FUNCTION_BLOCK Machine EXTENDS FB_PackML_BaseModule
VAR
	EquipOne	: EquipmentModule := (Name := 'Equip One');
	EquipTwo	: EquipmentModuleWithSubModule := (Name := 'Equip Two');
	ComponentMM : Component		  := (Name := 'Component MM');

	//Alarms
	MachineAlarms : ARRAY[1..MACHINE_ALARM_COUNT] OF FB_TcAlarm;
	testCritical  : BOOL;
	testError	  : BOOL;
	testWarning	  : BOOL;
	testInfo	  : BOOL;
	testVerbose	  : BOOL;
	clearAlarms	  : BOOL;
END_VAR

VAR CONSTANT
	MACHINE_ALARM_COUNT : UDINT := 6; //First is InitReferenceEvent
END_VAR

METHOD PROTECTED Clearing
VAR
	i				: UDINT;
	SubModulesReady : BOOL := TRUE;
	ComponentsReady : BOOL := TRUE;
END_VAR
(*
If there are no Components of the Machine
then we can clear the Machine Alarms and let the SUPER handle the rest.

But if the Machine Module has a component
then the process of clearing the alarms 
must be handled in a slightly different manner.
This will prevent an existing alarm condition that is still TRUE
from being cleared and raised multiple times.
*)
IF NumberOfComponents = 0 THEN
	F_ClearAllEventsInClass(Alarms := MachineAlarms);
	SUPER^.Clearing();
ELSE
	CASE SequenceState OF
		0:
			F_ClearAllEventsInClass(Alarms := MachineAlarms);
			SequenceState := SequenceState + 10;

		10:
			FOR i := 1 TO NumberOfSubModules DO
				ipSubModules[i].StateCommand := ePMLCommand_Clear;
			END_FOR

			IF BaseAlarms[E_BaseAlarms.ComponentError].bRaised THEN
				BaseAlarms[E_BaseAlarms.ComponentError].Clear(0, 0);
			END_IF;

			IF BaseAlarms[E_BaseAlarms.SubModuleError].bRaised THEN
				BaseAlarms[E_BaseAlarms.SubModuleError].Clear(0, 0);
			END_IF;

			SequenceState := SequenceState + 10;

		20:
			FOR i := 1 TO NumberOfComponents DO
				IF Parameters_PackML_Base.RESET_COMPONENTS_WITHOUT_ERROR THEN
					ipComponents[i].Reset();
				ELSE
					IF ipComponents[i].Error THEN
						ipComponents[i].Reset();
					END_IF
				END_IF
			END_FOR

			FOR i := 1 TO NumberOfComponents DO
				ComponentsReady := ComponentsReady AND NOT ipComponents[i].Error;
			END_FOR

			IF ComponentsReady THEN
				SequenceState := SequenceState + 10;
			END_IF

		30:
			FOR i := 1 TO NumberOfSubModules DO
				SubModulesReady := SubModulesReady AND (ipSubModules[i].CurrentState = ePMLState_Stopped);
			END_FOR

			IF SubModulesReady AND (StateTasksComplete OR NoStateTasksToComplete) THEN
				NoStateTasksToComplete := TRUE;
				StateTasksComplete	   := FALSE;
				StateComplete();
			END_IF
	END_CASE
END_IF
END_METHOD

//! @summary Initializes event function blocks using this module's name
METHOD PROTECTED CreateEvents

//! @description This method is called by <c>Initialize()</c> as required
F_CreateAllEventsInClass(Alarms		:= MachineAlarms,
						 ClassSize	:= SIZEOF(TC_Events.MachineEvents),
						 pInitEvent := ADR(TC_EVENTS.MachineEvents.InitReferenceEvent),
						 Prefix		:= Name);

SUPER^.CreateEvents();
END_METHOD

//! @summary This method serves as the entry point for all underlying FB logic

//! @description This method should be called cyclically by descendant function blocks by invoking <c>SUPER^.CyclicLogic()</c>.  Alternatively, the contents of this method could be reimplemented entirely in which case a call to this method would not be necessary.
METHOD PUBLIC CyclicLogic
VAR
	i : UDINT;
END_VAR
IF NOT _InitComplete THEN
	_InitComplete := Initialize();
	RETURN;
END_IF

//AlarmHandling();
IF testVerbose AND NOT MachineAlarms[E_MachineEvents.VerboseEvent].bRaised THEN
	RaiseAlarm2Args(MachineAlarms[E_MachineEvents.VerboseEvent], 'Note 1', 'Note 2');
END_IF

IF testCritical AND NOT MachineAlarms[E_MachineEvents.CriticalEvent].bRaised THEN
	RaiseAlarm2Args(MachineAlarms[E_MachineEvents.CriticalEvent], 'Note 1', 'Note 2');
END_IF

//The MachineMonitor is based on the SubModuleMonitor, but is only monitors itself
MachineMonitor();

//
SUPER^.CyclicLogic();

(*
*
*		Code must be after SUPER^.CyclicLogic();
*
*)

(* Update alarm severity from this module *)
_CurrentAlarmSeverity := F_GetMaxSeverityRaised(Alarms := MachineAlarms, CurrentSeverity := _CurrentAlarmSeverity);
_Error				  := _CurrentAlarmSeverity >= TcEventSeverity.Error;


Trace(Message:='Test Mesage');
END_METHOD

//! @summary Basic module initialization logic
METHOD PROTECTED Initialize : BOOL;
VAR
	i						 : UDINT;
	varInfo					 : __SYSTEM.VAR_INFO;
	AllSubUnitsInitialized	 : BOOL := TRUE;
	AllComponentsInitialized : BOOL := TRUE;
END_VAR

//! @description This method is called by <c>CyclicLogic()</c> as required
Initialize := FALSE;
CASE DescendantSequenceState OF
	0:
		LogModeChanges	:= FALSE;
		LogStateChanges := FALSE;

		//Register Submodules
		RegisterSubmodule(EquipOne);
		RegisterSubmodule(EquipTwo);		
		RegisterComponent(ComponentMM);
		DescendantSequenceState := DescendantSequenceState + 10;

	10:
		IF SUPER^.Initialize() THEN
			Initialize := TRUE;
		END_IF
END_CASE
END_METHOD

METHOD MachineMonitor
VAR
	AlarmResponses : ARRAY[0..4] OF E_AlarmResponse; //Temporary response array	
	i			   : UDINT;
END_VAR
IF _CurrentState <> E_PMLState.ePMLState_Aborted AND _CurrentState <> E_PMLState.ePMLState_Aborting AND _CurrentState <> E_PMLState.ePMLState_Clearing AND _CurrentState <> E_PMLState.ePMLState_Stopped AND _CurrentState <> E_PMLState.ePMLState_Stopping THEN
	AlarmResponses := ParentResponseDefinitions;
	CASE AlarmResponses[_CurrentAlarmSeverity] OF
		E_AlarmResponse.Abort_ImmediateError:
			AbortImmediateError(Name, TRUE);

		E_AlarmResponse.Abort_Immediate:
			AbortImmediate();

		E_AlarmResponse.Stop_Immediate:
			StopImmediate();

		E_AlarmResponse.Stop_Controlled:
			StopControlled();

		E_AlarmResponse.Hold_Immediate:
			HoldImmediate();

		E_AlarmResponse.Hold_Controlled:
			HoldControlled();

		E_AlarmResponse.Suspend_Immediate:
			SuspendImmediate();

		E_AlarmResponse.Suspend_Controlled:
			SuspendControlled();

		E_AlarmResponse.NoResponse:
			;
	END_CASE
ELSIF _CurrentState = E_PMLState.ePMLState_Stopped OR _CurrentState = E_PMLState.ePMLState_Stopping THEN
	AlarmResponses := ParentResponseDefinitions;
	CASE AlarmResponses[CurrentAlarmSeverity] OF
		E_AlarmResponse.Abort_ImmediateError:
			AbortImmediateError(Name, TRUE);

		E_AlarmResponse.Abort_Immediate:
			AbortImmediate();

		E_AlarmResponse.NoResponse:
			;
	END_CASE
END_IF
END_METHOD

METHOD RaiseAlarm2Args
VAR_IN_OUT
	Alarm : FB_TcAlarm; //Alarm to be raised
END_VAR

VAR_INPUT
	String_1 : STRING; //First String Parameter (The Name of this component will be applied first automatically)
	String_2 : STRING; //Second String Parameter
END_VAR
F_RaiseAlarmWithStringParameters(Alarm	  := Alarm,
								 String_1 := Name,
								 String_2 := String_1,
								 String_3 := String_2);
END_METHOD

END_FUNCTION_BLOCK

(* stored: Version 1.1.0.1, ProductVersion 3.1.4024.13
   POU Machine: Id {66cc6e36-2ea9-4621-bedd-f5d531d191bf}, SpecialFunc None
   Method Clearing: Id {218ba0d7-e931-4a28-8ae7-0db360a35c2d}
   Method CreateEvents: Id {4ed9832e-c5dc-46d4-abe9-a51eb498396c}
   Method CyclicLogic: Id {e574dd6e-a801-487f-b62e-c8264bb86070}
   Method Initialize: Id {d1725bba-8b00-4347-8fac-2b2ca6e24462}
   Method MachineMonitor: Id {8c8dc412-6c16-4a57-b8c9-8674903aa98b}
   Method RaiseAlarm2Args: Id {106a700c-ae28-40c8-8dd9-a78e7098e9ff} *)
